PROGRAM HMI
VAR
	Feedback		: HmiFeedback;
	Control			: HmiControl;
	
	NULL			: PVOID;
	UdpIO			: UdpClient(3232258620, 50160, 50150, SIZEOF(Feedback), ADR(Feedback), SIZEOF(Control), ADR(Control));
	
END_VAR


Feedback.Feedback 	:=  REMOTE.Feedback;
Feedback.Control 	:=  REMOTE.Control;


UdpIO();

(*
IF hmi_counter <> hmi_counter_old THEN
	hmi_flag := 0;
	hmi_counter_old := hmi_counter;
ELSE
	hmi_flag := hmi_flag + 1;
END_IF
*)

END_PROGRAM

(* stored: Version 1.1.0.1, ProductVersion 3.1.4020.12
   POU HMI: Id {92c9e502-42e5-4c53-8e84-6f6172dad33a}, SpecialFunc None *)
